(*
A list implementation for managing `I_Arg`.  
*)
FUNCTION_BLOCK CompList
VAR_GENERIC CONSTANT
	nCap	: UDINT := 100;
END_VAR

IMPLEMENTS I_MutCompList

VAR
	_iList	: ARRAY[1..nCap] OF I_Component;
END_VAR

(*
Provides the maximum capacity of the list.
*)
PROPERTY Cap : UDINT
GET
Cap := nCap;
END_GET
END_PROPERTY

(*
Retrieves the `I_Component` at the specified index.  
Returns:
- `Ok` - Successfully retrieves the `I_Component`.
- `Err.Idx` - The specified index is out of bounds.
- `Err.InvRef` - Invalid output reference.
- `Err.Idx` - `iOut` = 0.
*)
METHOD Get : Result
VAR_INPUT
	nIndex		: UDINT;
	iOut		: REFERENCE TO I_Component;
END_VAR
IF nIndex > nCap OR nIndex = 0 THEN
	Get := Err.Idx;
	RETURN;	
END_IF

IF NOT __ISVALIDREF(iOut) THEN
	Get := Err.InvRef;
	RETURN;
END_IF

iOut := _iList[nIndex];
IF iOut <> 0 THEN
	Get := Ok;
ELSE
	Get := Err.NotFound;
END_IF
END_METHOD

(*
Adds, updates, or removes an argument in the list at the specified index.  
Return:
- `Ok` - Upon successfully adding, modifying, or removing an entry.
- `Err.Idx` - When attempting to modify an entry at an out-of-bounds index.
*)
METHOD Set : Result
VAR_INPUT
	iIn			: I_Component;
	nIndex		: UDINT;
END_VAR
IF nIndex > nCap OR nIndex = 0 THEN
	Set := Err.Idx;
	RETURN;	
END_IF

_iList[nIndex] := iIn;
Set := Ok;
END_METHOD

END_FUNCTION_BLOCK

(* stored: Version 1.1.0.1
   POU CompList: Id {ab0a7914-9ac4-41cb-a281-5d9e708234e4}, SpecialFunc None
   Property Cap: Id {a16011eb-eccf-4267-a3d9-5dda38aa8b01}
   Get Get: Id {4d225c82-253b-4ef0-b494-d33220e45dcb}
   Method Get: Id {f84861e2-0afd-46b7-8244-73ebc3fcdd54}
   Method Set: Id {6e175e97-5942-4516-887c-86db013eb6a3} *)
